FUNCTION_BLOCK FB_OutRobot_EmptyBoxMove_old EXTENDS FB_ObjectBase_V2
VAR_INPUT
//    Execute    :BOOL;   // True : This prog will start.
//    Abort      :BOOL;   // True : This prog will be abort.
//    Reset      :BOOL;   // True : This prog will be reset.
//    ObjectName :STRING; // Set this fb name(About it's action)
	INPUT            			   : REFERENCE TO ST_InputTable;
	Cylinder   					   : REFERENCE TO UNI_CylinderList;
	Motor      					   : REFERENCE TO UNI_MotorList;
	AutoMode_OutRobotMoveMove : st_AutoMode_ClampingBoxesJob;	
	Cylinders					   : REFERENCE TO ARRAY[0..1] OF FB_Cylinder;
	Clips						   : REFERENCE TO ARRAY[0..1] OF FB_Cylinder;
END_VAR

VAR_OUTPUT
//    Busy    :BOOL;        // True : This prog is running.
//    Done    :BOOL;        // True : Command has been executed.
//    Aborted :BOOL;        // True : This prog is aborted.
//    Error   :BOOL;        // True : This prog has an error.
//    ErrorID :UINT;       // Output ErrorID
//    Status  :T_MaxString; // Output this prog status by string(255bytes)
END_VAR

VAR
//    eState :E_MethodStatus_Basic;
//	uiExecutingStep : UDINT; // This var is used to been controll STATE_EXECUTING process.
//	uiResettingStep : UDINT;
//	uiAbortingStep : UDINT;
//	_Executed :BOOL; // Executing process completed.
//	_Error : BOOL; // FB has an error.
//	_ResetCompleted : BOOL; // FB resetting completed.
//	_AbortCompleted : BOOL; // FB aborting completed.
	//_Abort		: BOOL;
	strStatus	: STRING;
	uiResumeStep : UINT;
	tonTimeOut   :TON;
	tonTimeDelay   :TON;
	iWorkingIndex : INT;
	_UniqueErrorCode :STRING;	
	
	PickingPos	: ARRAY[0..1] OF ST_PositionTable;
	PlacingPos  : ARRAY[0..1] OF ST_PositionTable;
	PressCylinderOnI5			   : REFERENCE TO FB_Cylinder;
	bSyncPick	: BOOL;
	bSyncPlace	: BOOL;
	SensorOnConveyor		   : BIT;
	ConveyorMotor				   : REFERENCE TO FB_Motor;
	UseA	: BOOL;
	UseB	: BOOL;
END_VAR

A00_BasicUnits();
SUPER^.A10_StateControl();

ACTION A00_BasicUnits:
tonTimeOut(PT:=T#60S);
tonTimeDelay(PT:=T#1s);
END_ACTION

METHOD GetModelState
VAR_OUTPUT
    xDone    :BOOL;
    xBusy    :BOOL;
    xError   :BOOL;
    xAborted :BOOL;
    iErrorID :UDINT;
	UniqueErrorCode : STRING;
END_VAR
xDone    := Done;
xBusy    := Busy;
xError   := Error;
xAborted := Abort;
iErrorID := ErrorID;
UniqueErrorCode := THIS^.UniqueErrorCode;
END_METHOD

METHOD GetName : STRING
GetName := ObjectName;
END_METHOD

METHOD PRIVATE M_CheckCommand : BOOL
VAR_INPUT
END_VAR


M_CheckCommand := true;
END_METHOD

METHOD PRIVATE M_GetWorkingConditions : BOOL
VAR_INPUT
END_VAR
IF AutoMode_OutRobotMoveMove.ClampingInfo.UseClibA THEN
	PickingPos[0] :=FUN_GetPositionTableData('I',5,0);
	PlacingPos[0]:=FUN_GetPositionTableData('R',1,0);
	UseA :=TRUE;
END_IF

IF AutoMode_OutRobotMoveMove.ClampingInfo.UseClibB THEN
	PickingPos[1] :=FUN_GetPositionTableData('I',5,1);
	PlacingPos[1]:=FUN_GetPositionTableData('R',2,1);
	UseB := TRUE;
END_IF

IF PlacingPos[0].X_Pos =PlacingPos[1].X_Pos AND PlacingPos[0].Y_Pos = PlacingPos[1].Y_Pos AND UseA AND UseB  THEN
		bSyncPlace:=TRUE;
	ELSE
		bSyncPlace:=FALSE;	
END_IF
IF PickingPos[0].X_Pos =PickingPos[1].X_Pos AND PickingPos[0].Y_Pos = PickingPos[1].Y_Pos AND UseA AND UseB THEN
		bSyncPick:=TRUE;
	ELSE
		bSyncPick:=FALSE;	
END_IF

PressCylinderOnI5 REF= Cylinder.List.fbDifferentSizeCV_Press2;


ConveyorMotor REF= Motor.List.TransmitDifferentSideCV;
END_METHOD

METHOD PRIVATE M_RecoveryAllObjects : BOOL
VAR_INPUT
END_VAR
VAR 
	i : INT;
END_VAR
FOR i:=0 TO 1 DO
	IF Clips[i].xError THEN
		Clips[i].M_Reset();
		ELSE
		Clips[i].M_Retract();		
	END_IF
	IF Cylinders[i].xError THEN
	Cylinders[i].M_Reset();	
	ELSE
	Cylinders[i].M_Retract();	
	END_IF
END_FOR


IF arAxisCtrl_gb[AxisNo.OutRobot_X].Admin.Axis.Status.Error THEN

	arAxisCtrl_gb[AxisNo.OutRobot_X].Admin.ClearError:= TRUE;
ELSE
	arAxisCtrl_gb[AxisNo.OutRobot_X].Admin.ClearError:= FALSE;
END_IF

IF arAxisCtrl_gb[AxisNo.OutRobot_Y].Admin.Axis.Status.Error THEN

	arAxisCtrl_gb[AxisNo.OutRobot_Y].Admin.ClearError:= TRUE;
ELSE
	arAxisCtrl_gb[AxisNo.OutRobot_Y].Admin.ClearError:= FALSE;
END_IF
END_METHOD

METHOD  M_STATE_ABORTED
VAR_INPUT
END_VAR
ERROR :=TRUE;
Busy    := FALSE;
Aborted := TRUE;
Status := strStatus;

IF NOT Execute THEN
	eSTATE:=STATE_RESETTING;
END_IF

IF Execute AND Reset THEN
//	uiExecutingStep :=uiResumeStep;
	eSTATE:=STATE_EXECUTING;
END_IF
END_METHOD

METHOD  M_STATE_ABORTING
VAR_INPUT
END_VAR
VAR	 
 i : INT;
	bCylinderCheck: BOOL;
END_VAR
Error := TRUE;
CASE uiAbortingStep OF
	0 :
		bCylinderCheck :=TRUE;
		ConveyorMotor.M_MotorStop();
	
		FOR i :=0 TO 1 DO		
	    	Cylinders[i].M_Reset();
			Cylinders[i].M_Retract();
			bCylinderCheck:=bCylinderCheck AND Cylinders[i].InRearPosition;	
		END_FOR
		IF bCylinderCheck THEN		
			uiAbortingStep:=9999;
		END_IF
	9999:	_AbortCompleted:=TRUE;
END_CASE

IF _AbortCompleted THEN	
	eSTATE :=STATE_ABORTED;
END_IF
END_METHOD

METHOD  M_STATE_DONE
VAR_INPUT
END_VAR
Busy 	:= FALSE;
Done	:=TRUE;

IF NOT Execute THEN
	eSTATE:=STATE_RESETTING;
END_IF
END_METHOD

METHOD  M_STATE_DORMANT
VAR_INPUT
END_VAR
Busy            := FALSE;
Done            := FALSE;
Aborted         := FALSE;
Error           := FALSE;
ErrorID         := 0;
Status          := '';
_ResetCompleted := FALSE;
_Error          := FALSE;
_Executed       := FALSE;
_Abort	 :=FALSE;
strStatus :='FB_OutRobot_EmptyBoxMove: No Error';
uiExecutingStep :=uiResettingStep :=uiResumeStep :=0;
tonTimeOut.IN :=TRUE;
_UniqueErrorCode:='0';
iWorkingIndex :=0;
bSyncPlace := FALSE;
UseA := FALSE;
UseB :=FALSE;
IF Execute THEN
	eSTATE:=STATE_EXECUTING;
END_IF
END_METHOD

METHOD  M_STATE_ERROR
VAR_INPUT
END_VAR
ERROR   :=TRUE;
Busy	:=FALSE;
Status := strStatus;
IF __ISVALIDREF(ConveyorMotor) THEN
	ConveyorMotor.M_MotorStop();
END_IF
IF NOT Execute THEN	
eSTATE:=STATE_RESETTING;
END_IF
END_METHOD

METHOD  M_STATE_EXECUTING
VAR_INPUT
END_VAR
VAR_INST
	bMoveConveyorForward : BOOL;
	bMoveConveyorBackrward : BOOL;

END_VAR

VAR
	bCylinderCheck : BOOL := TRUE;
END_VAR
Busy :=TRUE;
SensorOnConveyor := INPUT.bDifferentSizeCV_BoxDetect5_Sensor;
IF bMoveConveyorForward THEN
	IF NOT ConveyorMotor.InBackWard THEN
		ConveyorMotor.M_MoveForward();
	END_IF
END_IF
IF bMoveConveyorBackrward THEN
	IF NOT ConveyorMotor.InForWard THEN
		ConveyorMotor.M_MoveBackward();
	END_IF
END_IF
CASE uiExecutingStep OF
	

0: //Idle
	bMoveConveyorForward:=FALSE;
	bMoveConveyorBackrward:=FALSE;
	tonTimeDelay.IN :=FALSE;
	tonTimeOut.IN := FALSE;
	iWorkingIndex :=0;
	M_GetWorkingConditions();
	
	
	M_RecoveryAllObjects();
	uiExecutingStep := 100;
	
100: //Check command
	
	IF PressCylinderOnI5.xError THEN
		PressCylinderOnI5.M_Reset();
	ELSE
		PressCylinderOnI5.M_Retract();
	END_IF
	
	IF M_CheckCommand() THEN
		uiExecutingStep:=200;
	END_IF
	
200: // Check No boxes turntable

	IF (UseA AND INPUT.bTurnTable_R1Detect_Sensor) OR (UseB AND INPUT.bTurnTable_R2Detect_Sensor) THEN
		_Abort:=TRUE;
		strStatus :='FB_OutRobot_EmptyBoxMove Step 200: Box On Turntable';
	ELSE
		IF UseA THEN
			iWorkingIndex :=0;
		ELSE
			iWorkingIndex :=1;	
		END_IF
		
		uiExecutingStep:=1000;	
	END_IF

	
1000: 
	// Move Conveyor
	// Move OutRobot to First clip picking	
	 //ConveyorMotor.M_MoveForward();
	 bMoveConveyorForward:=TRUE;
	arAxisCtrl_gb[AxisNo.OutRobot_X].PosMode.Position := PickingPos[iWorkingIndex].X_Pos;		
	arAxisCtrl_gb[AxisNo.OutRobot_Y].PosMode.Position := PickingPos[iWorkingIndex].Y_Pos;	
		IF ConveyorMotor.InForWard THEN
			uiExecutingStep:=1100;
		END_IF
		
1100://CheckSensor
	tonTimeDelay.IN:=SensorOnConveyor;
	
			
	IF tonTimeDelay.Q THEN
		tonTimeOut.IN :=FALSE;
		uiExecutingStep:=1200;
		tonTimeDelay.IN := FALSE;
		
	END_IF
	
	tonTimeOut.IN := TRUE;
	IF tonTimeOut.Q THEN
		tonTimeOut.IN :=FALSE;
		_Abort := TRUE;
		strStatus :='FB_OutRobot_EmptyBoxMove Step 1100: No Box on conveyor';
	END_IF

1200: //Press seconde box
	  PressCylinderOnI5.M_Extend();
	  IF PressCylinderOnI5.InFrontPosition THEN
		  tonTimeOut.IN :=FALSE;
		  uiExecutingStep:=1300;
	  END_IF
	  
	  	tonTimeOut.IN := TRUE;
	IF tonTimeOut.Q THEN
		tonTimeOut.IN :=FALSE;
		_Abort := TRUE;
		strStatus :='FB_OutRobot_EmptyBoxMove Step 1200: Block box on conveyor timeout';
	END_IF
	
1300: // Stop conveyor
	ConveyorMotor.M_MotorStop();
	bMoveConveyorForward:=FALSE;
	bMoveConveyorBackrward:=FALSE;
	IF ConveyorMotor.InStopped THEN
		 uiExecutingStep:=1400;
	END_IF

1400: // Check outRobot arrived
	IF		(arAxisStatus_gb[AxisNo.OutRobot_X].Admin._OpModeAck = ModePosAbs AND arAxisStatus_gb[AxisNo.OutRobot_X].Admin.CmdDone) 
	AND (arAxisStatus_gb[AxisNo.OutRobot_Y].Admin._OpModeAck = ModePosAbs AND arAxisStatus_gb[AxisNo.OutRobot_Y].Admin.CmdDone) 
	THEN
		tonTimeOut.IN :=FALSE;
		uiExecutingStep:=1500;
	END_IF	
	
	tonTimeOut.IN := TRUE;
	IF tonTimeOut.Q THEN
		tonTimeOut.IN :=FALSE;
		_Error := TRUE;
		strStatus :='FB_OutRobot_EmptyBoxMove Step 1400: Move robot to picking position timeout';
	END_IF
	
1500: //Clip Down Pick
	 Cylinders[iWorkingIndex].M_Extend();
	  IF Cylinders[iWorkingIndex].InFrontPosition THEN
		  tonTimeOut.IN :=FALSE;
		  uiExecutingStep:=1700;
	  END_IF
	
	 tonTimeOut.IN := TRUE;
	IF tonTimeOut.Q THEN
		tonTimeOut.IN :=FALSE;
		_Abort := TRUE;
		strStatus :='FB_OutRobot_EmptyBoxMove Step 1500: Cylinder pick down timeout';
	END_IF
	
1700: // Clip close Pick
	Clips[iWorkingIndex].M_Extend();
	  IF Clips[iWorkingIndex].InFrontPosition THEN
		  tonTimeOut.IN :=FALSE;
		  uiExecutingStep:=1800;
	  END_IF
	  
	   tonTimeOut.IN := TRUE;
	IF tonTimeOut.Q THEN
		tonTimeOut.IN :=FALSE;
		_Abort := TRUE;
		strStatus :='FB_OutRobot_EmptyBoxMove Step 1700: clip pick close timeout';
	END_IF

1800: // Clip Up Pick
	   Cylinders[iWorkingIndex].M_Retract();
	  IF Cylinders[iWorkingIndex].InRearPosition THEN
		  
		  tonTimeOut.IN :=FALSE;
		  uiExecutingStep:=1850;
	  END_IF
	  
	    tonTimeOut.IN := TRUE;
	IF tonTimeOut.Q THEN
		tonTimeOut.IN :=FALSE;
		_Abort := TRUE;
		strStatus :='FB_OutRobot_EmptyBoxMove Step 1800: cylinder pick up timeout';
	END_IF
1850: //Check box leave
		IF NOT SensorOnConveyor THEN
			PressCylinderOnI5.M_Retract();
			uiExecutingStep:=1900;
		else
			_Error := TRUE;
			strStatus :='FB_OutRobot_EmptyBoxMove Step 1850: Box still on conveyor';
		END_IF
		
1900: // If Next pick
	  IF iWorkingIndex>=1 OR NOT UseB THEN
		  IF UseA THEN
		  	iWorkingIndex :=0;
		  ELSIF UseB THEN
			iWorkingIndex :=1;	
		  END_IF
		  uiExecutingStep:=2000;
		  //Go to placing box
	  ELSIF  iWorkingIndex=0 AND UseB THEN
			iWorkingIndex:=iWorkingIndex+1;
	 		uiExecutingStep:=1000;
	  END_IF
	  
2000: // Move to Placing pos
	 arAxisCtrl_gb[AxisNo.OutRobot_X].PosMode.Position := PlacingPos[iWorkingIndex].X_Pos;		
	 arAxisCtrl_gb[AxisNo.OutRobot_Y].PosMode.Position := PlacingPos[iWorkingIndex].Y_Pos;	
	 uiExecutingStep:=2100;

2100: // Waiting outRobot move to placing pos	 
	 IF	(arAxisStatus_gb[AxisNo.OutRobot_X].Admin._OpModeAck = ModePosAbs AND arAxisStatus_gb[AxisNo.OutRobot_X].Admin.CmdDone) 
	AND (arAxisStatus_gb[AxisNo.OutRobot_Y].Admin._OpModeAck = ModePosAbs AND arAxisStatus_gb[AxisNo.OutRobot_Y].Admin.CmdDone) 
	THEN
		tonTimeOut.IN :=FALSE;
		uiExecutingStep:=2200;
	END_IF	

	    tonTimeOut.IN := TRUE;
	IF tonTimeOut.Q THEN
		tonTimeOut.IN :=FALSE;
		_Error := TRUE;
		strStatus :='FB_OutRobot_EmptyBoxMove Step 2100: Move robot to placing position timeout';
	END_IF
	
2200: //Cllp Down place
	bCylinderCheck := TRUE;
	Cylinders[iWorkingIndex].M_Extend();
	bCylinderCheck :=Cylinders[iWorkingIndex].InFrontPosition AND bCylinderCheck;
	IF bSyncPlace THEN
		Cylinders[1].M_Extend();
		bCylinderCheck :=Cylinders[1].InFrontPosition AND bCylinderCheck;
	END_IF	
	 
	IF bCylinderCheck THEN
		tonTimeOut.IN :=FALSE;
		uiExecutingStep:=2300;
	END_IF 
	
	   tonTimeOut.IN := TRUE;
	IF tonTimeOut.Q THEN
		tonTimeOut.IN :=FALSE;
		_Abort := TRUE;
		strStatus :='FB_OutRobot_EmptyBoxMove Step 2200: Cylinder place down timeout';
	END_IF
	
2300: // Clip open Place
	bCylinderCheck := TRUE;
	Clips[iWorkingIndex].M_Retract();
	bCylinderCheck := Clips[iWorkingIndex].InRearPosition AND bCylinderCheck;
	IF bSyncPlace THEN
		Clips[1].M_Retract();
		bCylinderCheck := Clips[1].InRearPosition AND bCylinderCheck;
	END_IF	
	 
	IF bCylinderCheck THEN
		tonTimeOut.IN :=FALSE;
		uiExecutingStep:=2400;
	END_IF 
	  
	  tonTimeOut.IN := TRUE;
	IF tonTimeOut.Q THEN
		tonTimeOut.IN :=FALSE;
		_Abort := TRUE;
		strStatus :='FB_OutRobot_EmptyBoxMove Step 2300: clip place open timeout';
	END_IF
	  
2400: // Clip up Placing
	bCylinderCheck := TRUE;
	Cylinders[iWorkingIndex].M_Retract();
	bCylinderCheck :=Cylinders[iWorkingIndex].InRearPosition AND bCylinderCheck;
	IF bSyncPlace THEN
		Cylinders[1].M_Retract();
		bCylinderCheck :=Cylinders[1].InRearPosition AND bCylinderCheck;
	END_IF	
	 
	IF bCylinderCheck THEN
		tonTimeOut.IN :=FALSE;
		uiExecutingStep:=2500;
	END_IF 
	  tonTimeOut.IN := TRUE;
	IF tonTimeOut.Q THEN
		tonTimeOut.IN :=FALSE;
		_Abort := TRUE;
		strStatus :='FB_OutRobot_EmptyBoxMove Step 2400: cylinder place up timeout';
	END_IF
	
2500: // If Next place
	IF iWorkingIndex>=1 OR bSyncPlace OR NOT UseB THEN
		uiExecutingStep:=2600;
		// Finish
	ELSE	
		iWorkingIndex := iWorkingIndex+1;
	  	uiExecutingStep:=2000;
	END_IF
2600: //Check box on turntable

	IF (UseA AND NOT INPUT.bTurnTable_R1Detect_Sensor) OR (UseB AND NOT INPUT.bTurnTable_R2Detect_Sensor) THEN
		_Error:=TRUE;
		strStatus :='FB_OutRobot_EmptyBoxMove Step 2600: Box not On Turntable';
	ELSE
		uiExecutingStep:=3000;
	END_IF
3000: // Finish	
	bMoveConveyorForward:=FALSE;
	bMoveConveyorBackrward:=FALSE;
	_Executed:=TRUE;
	
END_CASE
	
IF NOT Execute THEN
	eState:=STATE_RESETTING;
END_IF
IF _Error THEN
	eState:=STATE_ERROR;
END_IF
IF _Abort THEN
	eSTATE:=STATE_ABORTING;
END_IF
IF _Executed THEN
	eSTATE:=STATE_Done;
END_IF
END_METHOD

METHOD  M_STATE_RESETTING
VAR_INPUT
END_VAR
Error :=_Error;
Done :=_Executed;
Busy := FALSE;


CASE uiResettingStep OF
	
	0:
		uiResettingStep:=9999;
		ConveyorMotor.M_MotorStop();
		M_RecoveryAllObjects();
		IF PressCylinderOnI5.xError THEN
		PressCylinderOnI5.M_Reset();
	ELSE
		PressCylinderOnI5.M_Retract();
	END_IF

	9999:
		_ResetCompleted:=TRUE;
END_CASE
IF _ResetCompleted THEN
	eSTATE:=STATE_DORMANT;
END_IF
END_METHOD

END_FUNCTION_BLOCK

(* stored: Version 1.1.0.1, ProductVersion 3.1.4024.13
   POU FB_OutRobot_EmptyBoxMove_old: Id {3d035ba1-18da-45db-9028-9ceb0a0d377b}, SpecialFunc None
   Folder Method: Id {bb6434ce-4d3c-4ebe-97cf-b00de6720102}
   Folder STATE: Id {df840c99-e90c-43c9-9ce4-0e451c67e8fc}
   Action A00_BasicUnits: Id {5c4a0465-3231-45f9-b78b-41a504520151}
   Method GetModelState: Id {9486c039-b902-4600-823c-e1475b25a352}
   Method GetName: Id {b1d59d9a-7307-463b-b4b8-c5cd7c94cf9d}
   Method M_CheckCommand: Id {5b8e0f0f-77b0-4457-a12c-a7b6d1b30424}
   Method M_GetWorkingConditions: Id {6ce36352-2975-4eb9-a664-c6341358856f}
   Method M_RecoveryAllObjects: Id {0ff61988-539e-4c92-971e-b9e14798b1de}
   Method M_STATE_ABORTED: Id {25f8093f-5b28-49ae-bfb2-c88e671ed144}
   Method M_STATE_ABORTING: Id {71f50659-aed8-411a-a365-80d9c7e3f473}
   Method M_STATE_DONE: Id {b8674a28-fd11-455c-a7b3-d1b16fced56f}
   Method M_STATE_DORMANT: Id {8d871cfe-d4d8-46f9-b68a-1c0dcfc0879e}
   Method M_STATE_ERROR: Id {e5328cb3-282e-49e9-9e35-d0080dc40854}
   Method M_STATE_EXECUTING: Id {1d7ae400-7c76-4840-9122-1dc2f3da695c}
   Method M_STATE_RESETTING: Id {2db424f0-ef6c-4eef-834c-dc81219a1369} *)
